PROGRAM MAIN
VAR
	iTest AT %I* : INT;
	iTest2 : INT := 0;
	
	iKlemme AT %I* : USINT;
	iOut AT %Q* : USINT;
END_VAR

iTest2 := iKlemme;

iOut := iKlemme;

END_PROGRAM

(* stored: Version 1.1.0.1, ProductVersion 3.1.4024.12
   POU MAIN: Id {c0a909f1-bd32-4d83-9fa7-8f7919b7094f}, SpecialFunc None *)
